Staubli VAL3: stopMotion.pgx

public program stopMotion()
begin
  // stop the motion using an event
  if cycleStatus:bStop==false
    setMutex(cycleStatus:bMotionToken)
    logMsg("[KERNEL] CYCLE:Stop motion")
    // enable the bit
    cycleStatus:bStop=true
    stopMove()
    // check that the robot has been stopped
    if watch(cycleStatus:bMoveStopped==true,10)==false
      logMsg("error stopping the robot using an INPUT ")
      wait(cycleStatus:bMoveStopped==true)
    endIf
  endIf
end
